ABB RobotStudio station: TransferLab2_final.rspag

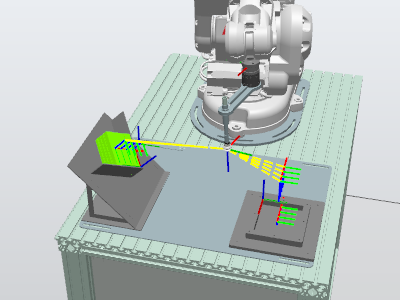
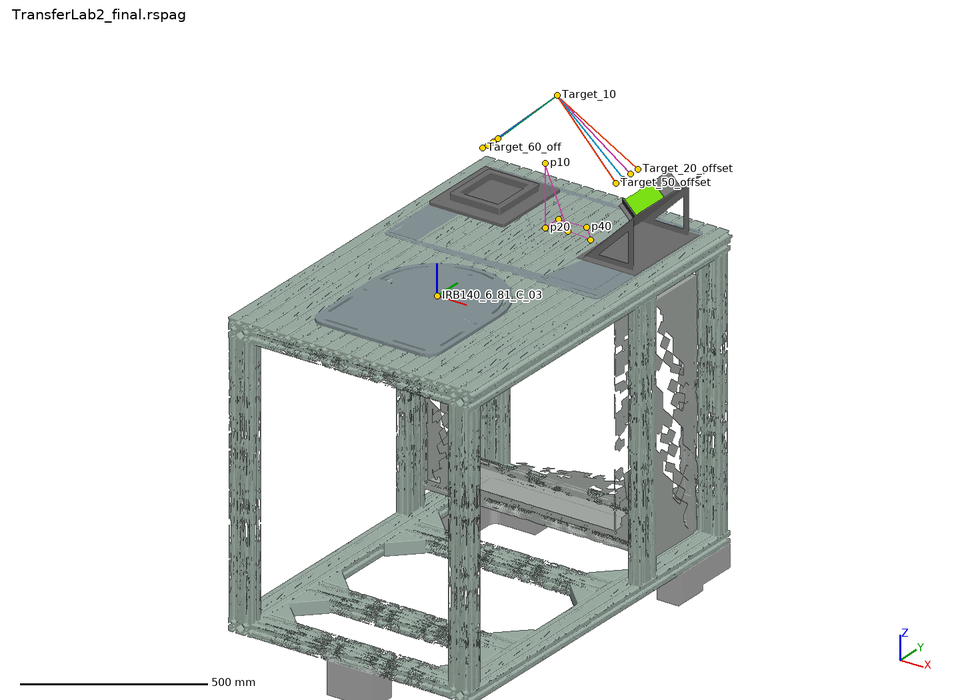
[picture v1: parts stored in the station drawn from their meshes, with robot base, taught points and paths (robot models come from the ABB library and are not in the file)]
--- station ---
Station AdvancedPickandPlace (saved by RobotStudio 24.1.10713.1)
Controller 140-107610, task T_ROB1: task frame (RAPID world) sits at (355.04, -190.94, 920) mm, rotated rx 0 ry 0 rz 90 deg in the station
Controller 140-107610
  mechanical unit ROB_1: IRB140_6_81_C_03, 6 joints, base frame (0, 0, 0) mm
Layout (positions relative to the parent item):
  - IRB140_6_81_C_03 [mechanism, from %ABB.RobotStudio.Models.IRB140%\IRB140_6_81_C_G_03.rslib] at (355.04, -190.94, 920) mm, rotated rx 0 ry 0 rz 90 deg; joint values [0.1928, 0.3139, 0.0677, 0.0702, 1.1676, -2.716] (rad or m)
  - Tpencil_2 [mechanism, from Libraries\Tpencil.rslib] at (0, 0, 0) mm
  - Modul_Base.prt [part], size 803.5 x 1200 x 1040 mm
  - FixturV [part] at (133.21, 403.34, 913) mm, size 245 x 265 x 30 mm
  - SnedLager_2 [part] at (709.45, 222.16, 913) mm, rotated rx 0 ry 0 rz 90 deg, size 300.2 x 214.3 x 218.7 mm
  - IRC5_Singel-Cabinet_2 [part, from %ABB.RobotStudio.Models.IRC5%\IRC5_Single-Cabinet.rslib] at (506.33, -200.93, 45.49) mm, rotated rx 90 ry 0 rz 90 deg
  - AE 1077.500 (2) [part] at (361.97, 363.55, 68.84) mm, rotated rx 90 ry 0 rz 180 deg, size 760 x 760 x 217 mm
  - tVacuum [mechanism, from Libraries\tVacuum.rslib] at (248.37, 333.62, 1408.02) mm, rotated rx -176.11 ry 0.46 rz 75.14 deg
  - SmartComponent_1 [smart component]
    - Source [smart component, from Components\Source.rslib]
        properties: Source=(none); Copy=cuboid_black_16; Parent=(none); Position=[0 0 0]; Orientation=[0 0 0]; Transient=false; PhysicsBehavior=0
  - cuboid_black_1 [part] at (1319.88, -207.47, 357.2) mm, rotated rx -33.6 ry -27.27 rz 53.23 deg, size 23.4 x 118 x 15.7 mm
  - cuboid_black_2 [part] at (1331.4, -191.2, 368.68) mm, rotated rx -33.6 ry -27.27 rz 53.23 deg, size 23.4 x 118 x 15.7 mm
  - cuboid_black_3 [part] at (1342.92, -174.94, 380.16) mm, rotated rx -33.6 ry -27.27 rz 53.23 deg, size 23.4 x 118 x 15.7 mm
  - cuboid_black_4 [part] at (1354.44, -158.68, 391.64) mm, rotated rx -33.6 ry -27.27 rz 53.23 deg, size 23.4 x 118 x 15.7 mm
  - cuboid_black_5 [part] at (1310.35, -207.47, 366.76) mm, rotated rx -33.6 ry -27.27 rz 53.23 deg, size 23.4 x 118 x 15.7 mm
  - cuboid_black_6 [part] at (1321.87, -191.2, 378.24) mm, rotated rx -33.6 ry -27.27 rz 53.23 deg, size 23.4 x 118 x 15.7 mm
  - cuboid_black_7 [part] at (1333.39, -174.94, 389.72) mm, rotated rx -33.6 ry -27.27 rz 53.23 deg, size 23.4 x 118 x 15.7 mm
  - cuboid_black_8 [part] at (1344.91, -158.68, 401.2) mm, rotated rx -33.6 ry -27.27 rz 53.23 deg, size 23.4 x 118 x 15.7 mm
  - cuboid_black_9 [part] at (1300.82, -207.47, 376.32) mm, rotated rx -33.6 ry -27.27 rz 53.23 deg, size 23.4 x 118 x 15.7 mm
  - cuboid_black_10 [part] at (1312.34, -191.2, 387.8) mm, rotated rx -33.6 ry -27.27 rz 53.23 deg, size 23.4 x 118 x 15.7 mm
  - cuboid_black_11 [part] at (1323.86, -174.94, 399.28) mm, rotated rx -33.6 ry -27.27 rz 53.23 deg, size 23.4 x 118 x 15.7 mm
  - cuboid_black_12 [part] at (1335.38, -158.68, 410.76) mm, rotated rx -33.6 ry -27.27 rz 53.23 deg, size 23.4 x 118 x 15.7 mm
  - cuboid_black_13 [part] at (1295.8, -202.6, 389.58) mm, rotated rx -33.76 ry -27.57 rz 53.58 deg, size 23.4 x 118 x 15.7 mm
  - cuboid_black_14 [part] at (1302.81, -191.2, 397.36) mm, rotated rx -33.6 ry -27.27 rz 53.23 deg, size 23.4 x 118 x 15.7 mm
  - cuboid_black_15 [part] at (1314.33, -174.94, 408.84) mm, rotated rx -33.6 ry -27.27 rz 53.23 deg, size 23.4 x 118 x 15.7 mm
  - cuboid_black_16 [part] at (1325.85, -158.68, 420.32) mm, rotated rx -33.6 ry -27.27 rz 53.23 deg, size 23.4 x 118 x 15.7 mm
  - RobotFrame [frame] at (355.04, -263.33, 920) mm, rotated rx 0 ry 0 rz 90 deg
Attachment: tVacuum is attached to IRB140_6_81_C_03 / Link6
Attachment: DropBox is attached to FixturV
Attachment: InclinedPickupBox is attached to SnedLager_2
Attachment: WobjTable is attached to Modul_Base.prt
EventTableEntry 1817: Group=, Trigger=doValve1 1818, Actions=[EventTableActionAttach 1819], Comment=, ActivationMode=2, Cyclic=false
EventTableTriggerIO 1818: IOValue=[1], IRC5Controller=? -1, Operator=0, SignalSource=140-107610 514
EventTableActionAttach 1819: AttachmentParent=tVacuum 1615, AttachmentChild=? -1, MountObject=false, Offset=[X=1, Y=0, Z=0, W=0, X=0, Y=1, Z=0, W=0, X=0, Y=0, Z=1, W=0, X=0, Y=0, Z=0, W=1], FlangeIndext=0, FindNearest=true
EventTableEntry 1820: Group=, Trigger=doValve1 1821, Actions=[EventTableActionDetach 1822], Comment=, ActivationMode=2, Cyclic=false
EventTableTriggerIO 1821: IOValue=[0], IRC5Controller=? -1, Operator=0, SignalSource=140-107610 514
EventTableActionDetach 1822: AttachmentParent=tVacuum 1615, AttachmentChild=? -1

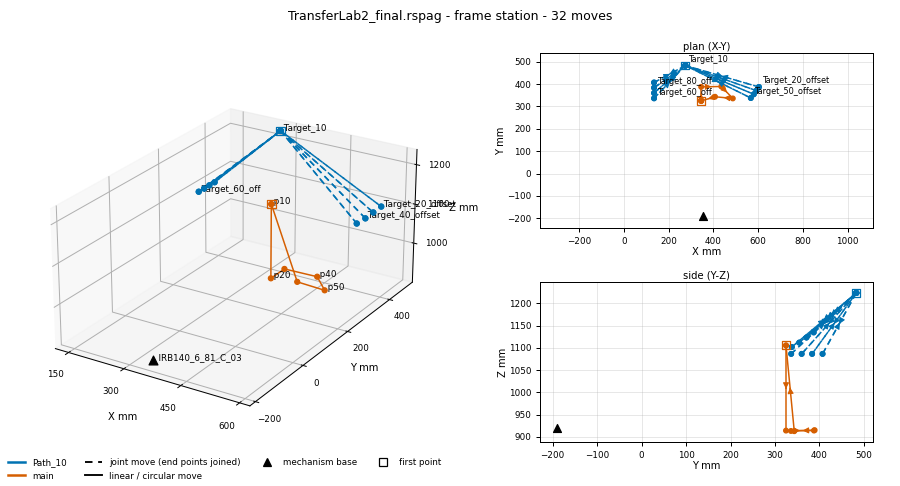
[picture p0: tool path of TransferLab2_final.rspag in frame station, 32 of 40 moves have a stored position in this frame; points joined in program order, loops and branches not executed]
--- Backups/140-107610/RAPID/TASK1/PROGMOD/MainModule.mod ---
MODULE MainModule
    PERS tooldata tVacuum:=[TRUE,[[152.46,0,183.744],[0,0,0,1]],[1.1,[1.547,-22.709,50.681],[1,0,0,0],0,0,0]];
    TASK PERS wobjdata WobjTable:=[FALSE,TRUE,"",[[280.944,-314.407,-7],[1,0,0,0]],[[0,0,0],[1,0,0,0]]];
    TASK PERS wobjdata InclinedPickupBox:=[FALSE,TRUE,"",[[562.907,-210.848,111.898],[0.35368,-0.146141,-0.352817,-0.853858]],[[0,0,0],[1,0,0,0]]];
    TASK PERS wobjdata DropBox:=[FALSE,TRUE,"",[[511.185,160.593,23],[1,0,0,0]],[[0,0,0],[1,0,0,0]]];
    !VAR intnum offset:= 14;
    !VAR intnum offset_z1;
    !VAR intnum offset_z2;
    PERS num countar :=1;



    PROC main()

        !FOR i  FROM 1 TO 5 DO
        !    offset :=14 * (i-1);
        !    offset_z1 := offset;
        !    offset_z2 := -1*offset;
        !ENDFOR

        Path_10;

    ENDPROC
ENDMODULE

--- Backups/140-107610/RAPID/TASK1/PROGMOD/Module1.mod ---
MODULE Module1
    CONST robtarget Target_10:=[[392.746094687,394.395276099,310.477856879],[0.000402904,0.129403902,0.991003532,0.034153585],[0,0,-2,0],[9E+09,9E+09,9E+09,9E+09,9E+09,9E+09]];

    CONST robtarget Target_20:=[[59.031543878,80.602128805,-4.00271589],[0.008197421,0.716388228,-0.697647201,-0.003015209],[-1,-1,-1,0],[9E+09,9E+09,9E+09,9E+09,9E+09,9E+09]];
    CONST robtarget Target_30:=[[59.031199796,57.602433832,-4.002496965],[0.008197421,0.716388228,-0.697647201,-0.003015209],[0,-1,-1,0],[9E+09,9E+09,9E+09,9E+09,9E+09,9E+09]];
    CONST robtarget Target_40:=[[59.031063684,34.601532617,-4.002986367],[0.008197421,0.716388228,-0.697647201,-0.003015209],[0,-1,-1,0],[9E+09,9E+09,9E+09,9E+09,9E+09,9E+09]];
    CONST robtarget Target_50:=[[59.260679093,11.297227236,-1.68849431],[0.008197421,0.716388228,-0.697647201,-0.003015209],[0,-1,-1,0],[9E+09,9E+09,9E+09,9E+09,9E+09,9E+09]];
    CONST robtarget Target_20_offset:=[[59.819440683,80.979027184,45.98965519],[0.008197421,0.716388228,-0.697647201,-0.003015209],[-1,-1,-1,0],[9E+09,9E+09,9E+09,9E+09,9E+09,9E+09]];
    CONST robtarget Target_30_offset:=[[59.819096601,57.979332211,45.989874115],[0.008197421,0.716388228,-0.697647201,-0.003015209],[0,-1,-1,0],[9E+09,9E+09,9E+09,9E+09,9E+09,9E+09]];
    CONST robtarget Target_40_offset:=[[59.818960489,34.978430996,45.989384713],[0.008197421,0.716388228,-0.697647201,-0.003015209],[-1,-1,-1,0],[9E+09,9E+09,9E+09,9E+09,9E+09,9E+09]];
    CONST robtarget Target_50_offset:=[[60.048575898,11.674125615,48.30387677],[0.008197421,0.716388228,-0.697647201,-0.003015209],[0,-1,-1,0],[9E+09,9E+09,9E+09,9E+09,9E+09,9E+09]];

    CONST robtarget Target_60:=[[16.076668507,59.018,-6.54],[0,0,1,0],[0,0,-2,0],[9E+09,9E+09,9E+09,9E+09,9E+09,9E+09]];
    CONST robtarget Target_60_off:=[[16.076668507,59.018,143.46],[0,0,1,0],[0,0,-2,0],[9E+09,9E+09,9E+09,9E+09,9E+09,9E+09]];
    CONST robtarget Target_70:=[[39.676668507,59.018,-6.54],[0,0,1,0],[0,0,-2,0],[9E+09,9E+09,9E+09,9E+09,9E+09,9E+09]];
    CONST robtarget Target_70_off:=[[39.676668507,59.018,143.46],[0,0,1,0],[0,0,-2,0],[9E+09,9E+09,9E+09,9E+09,9E+09,9E+09]];
    CONST robtarget Target_80:=[[63.176668507,59.018,-6.54],[0,0,1,0],[0,0,-2,0],[9E+09,9E+09,9E+09,9E+09,9E+09,9E+09]];
    CONST robtarget Target_80_off:=[[63.176668507,59.018,143.46],[0,0,1,0],[0,0,-2,0],[9E+09,9E+09,9E+09,9E+09,9E+09,9E+09]];
    CONST robtarget Target_90:=[[86.676668507,59.018,-6.54],[0,0,1,0],[0,0,-2,0],[9E+09,9E+09,9E+09,9E+09,9E+09,9E+09]];
    CONST robtarget Target_90_off:=[[86.676668507,59.018,143.46],[0,0,1,0],[0,0,-2,0],[9E+09,9E+09,9E+09,9E+09,9E+09,9E+09]];
    VAR intnum offset;
    VAR intnum offset_z1;
    VAR intnum offset_z2;


    PROC Path_10()

        FOR i  FROM 0 TO 3 DO
            offset :=14 * i;
            offset_z1 := -1*offset;
            offset_z2 := offset;

            MoveJ Target_10,v200,fine,tVacuum\WObj:=WobjTable;
            MoveJ Target_20_offset,v200,fine,tVacuum\WObj:=InclinedPickupBox;
            MoveJ Offs(Target_20,0,0,offset_z1),v200,fine,tVacuum\WObj:=InclinedPickupBox;
            !MoveJ Target_20,v200,fine,tVacuum\WObj:=InclinedPickupBox;
            WaitTime 0.3;
            SetDO doValve1, 1;
            WaitTime 0.3;
            MoveJ Target_20_offset,v200,fine,tVacuum\WObj:=InclinedPickupBox;
            MoveJ Target_10,v200,fine,tVacuum\WObj:=WobjTable;
            MoveJ Target_60_off,v200,fine,tVacuum\WObj:=DropBox;
            MoveJ Offs(Target_60,0,0,offset_z2),v200,fine,tVacuum\WObj:=DropBox;
            !MoveJ Target_60,v200,fine,tVacuum\WObj:=DropBox;
            WaitTime 0.3;
            SetDO doValve1, 0;
            WaitTime 0.3;
            MoveJ Target_60_off,v200,fine,tVacuum\WObj:=DropBox;

            MoveJ Target_10,v200,fine,tVacuum\WObj:=WobjTable;
            MoveJ Target_30_offset,v200,fine,tVacuum\WObj:=InclinedPickupBox;
            MoveJ Offs(Target_30,0,0,offset_z1),v200,fine,tVacuum\WObj:=InclinedPickupBox;
            WaitTime 0.3;
            SetDO doValve1, 1;
            WaitTime 0.3;
            MoveJ Target_30_offset,v200,fine,tVacuum\WObj:=InclinedPickupBox;
            MoveJ Target_10,v200,fine,tVacuum\WObj:=WobjTable;
            MoveJ Target_70_off,v200,fine,tVacuum\WObj:=DropBox;
            MoveJ Offs(Target_70,0,0,offset_z2),v200,fine,tVacuum\WObj:=DropBox;
            WaitTime 0.3;
            SetDO doValve1, 0;
            WaitTime 0.3;
            MoveJ Target_70_off,v200,fine,tVacuum\WObj:=DropBox;

            MoveJ Target_10,v200,fine,tVacuum\WObj:=WobjTable;
            MoveJ Target_40_offset,v200,fine,tVacuum\WObj:=InclinedPickupBox;
            MoveJ Offs(Target_40,0,0,offset_z1),v200,fine,tVacuum\WObj:=InclinedPickupBox;
            WaitTime 0.3;
            SetDO doValve1, 1;
            WaitTime 0.3;
            MoveJ Target_40_offset,v200,fine,tVacuum\WObj:=InclinedPickupBox;
            MoveJ Target_10,v200,fine,tVacuum\WObj:=WobjTable;
            MoveJ Target_80_off,v200,fine,tVacuum\WObj:=DropBox;
            MoveJ Offs(Target_80,0,0,offset_z2),v200,fine,tVacuum\WObj:=DropBox;
            WaitTime 0.3;
            SetDO doValve1, 0;
            WaitTime 0.3;
            MoveJ Target_80_off,v200,fine,tVacuum\WObj:=DropBox;

            MoveJ Target_10,v200,fine,tVacuum\WObj:=WobjTable;
            MoveJ Target_50_offset,v200,fine,tVacuum\WObj:=InclinedPickupBox;
            MoveJ Offs(Target_50,0,0,offset_z1),v200,fine,tVacuum\WObj:=InclinedPickupBox;
            WaitTime 0.3;
            SetDO doValve1, 1;
            WaitTime 0.3;
            MoveJ Target_50_offset,v200,fine,tVacuum\WObj:=InclinedPickupBox;
            MoveJ Target_10,v200,fine,tVacuum\WObj:=WobjTable;
            MoveJ Target_90_off,v200,fine,tVacuum\WObj:=DropBox;
            MoveJ Offs(Target_90,0,0,offset_z2),v200,fine,tVacuum\WObj:=DropBox;
            WaitTime 0.3;
            SetDO doValve1, 0;
            WaitTime 0.3;
            MoveJ Target_90_off,v200,fine,tVacuum\WObj:=DropBox;
            MoveJ Target_10,v200,fine,tVacuum\WObj:=WobjTable;

        ENDFOR


    ENDPROC
ENDMODULE

--- Backups/140-107610/HOME/wobj1/MainModule.mod ---
MODULE MainModule
	PERS tooldata tpencil:=[TRUE,[[-158.365,-2.10512,218.153],[1,0,0,0]],[0.5,[0,50,20],[1,0,0,0],0,0,0]];
	CONST robtarget p10:=[[515.61,9.13,185.47],[0.0619205,-0.079314,-0.994803,-0.0155883],[0,0,4,0],[9E+09,9E+09,9E+09,9E+09,9E+09,9E+09]];
	CONST robtarget p20:=[[515.61,9.13,-6.06],[0.0619228,-0.0793163,-0.994802,-0.0155846],[0,0,4,0],[9E+09,9E+09,9E+09,9E+09,9E+09,9E+09]];
	CONST robtarget p30:=[[578.43,9.13,-5.93],[0.0619495,-0.0792905,-0.994803,-0.015573],[0,0,4,0],[9E+09,9E+09,9E+09,9E+09,9E+09,9E+09]];
	CONST robtarget p40:=[[580.05,-80.82,-5.11],[0.0619285,-0.0793003,-0.994803,-0.0155876],[-1,0,3,0],[9E+09,9E+09,9E+09,9E+09,9E+09,9E+09]];
	CONST robtarget p50:=[[526.72,-132.09,-6.90],[0.0619458,-0.0792925,-0.994803,-0.0155861],[-1,0,3,0],[9E+09,9E+09,9E+09,9E+09,9E+09,9E+09]];
	CONST robtarget p60:=[[534.19,-52.76,-7.42],[0.0619566,-0.0792931,-0.994802,-0.015582],[-1,0,4,0],[9E+09,9E+09,9E+09,9E+09,9E+09,9E+09]];
	CONST robtarget p80:=[[533.93,-53.00,-9.15],[0.0619823,-0.0792257,-0.994806,-0.0155703],[-1,0,4,0],[9E+09,9E+09,9E+09,9E+09,9E+09,9E+09]];
	TASK PERS wobjdata wobj1:=[FALSE,TRUE,"",[[437.294,-191.242,-5.21685],[0.999806,-0.00979503,0.0148767,0.00835695]],[[0,0,0],[1,0,0,0]]];
	TASK PERS wobjdata wobj2:=[FALSE,TRUE,"",[[560.405,50.3251,-9.50006],[0.999834,0.00238531,-0.015124,0.00988946]],[[0,0,0],[1,0,0,0]]];
	PROC main()
		MoveJ p10, v300, fine, tpencil;
		MoveL p20, v300, fine, tpencil;
		MoveL p30, v300, fine, tpencil;
		MoveL p40, v300, fine, tpencil;
		MoveL p50, v300, fine, tpencil;
		MoveL p60, v300, fine, tpencil;
		MoveL p10, v300, fine, tpencil;
	ENDPROC
ENDMODULE

--- Backups/140-107610/SYSPAR/EIO.cfg ---
EIO:CFG_1.0:6:1::
#
SYSSIG_OUT:

      -Status "MotorOn" -Signal "doMotorLamp"

      -Status "EmStop" -Signal "doEmstopLamp"
#
INDUSTRIAL_NETWORK:

      -Name "DeviceNet" -Label "DeviceNet Master/Slave Network" -Address "2"

      -Name "PROFIBUS_Anybus" -Label "PROFIBUS Anybus Network" -Address "125"
#
EIO_CROSS:

      -Name "SYJ5325Control1" -Res "doSYJ5323_A" -Act1 "doValve1" -Oper1 "AND"\
      -Act2 "doYJ5123" -Act2_invert

      -Name "SYJ5323Control2" -Res "doSYJ5323_B" -Act1 "doValve1" -Act1_invert \
      -Oper1 "AND" -Act2 "doYJ5123" -Act2_invert

      -Name "SYJ5123Control" -Res "doYJ5123" -Act1 "diToolChangeButton"\
      -Oper1 "OR" -Act2 "doToolChanger"
#
ETHERNETIP_DEVICE:

      -Name "Local_IO" -VendorName "ABB Robotics" -ProductName "DSQC1030"\
      -Label "ABB Local I/O Device" -Address "192.168.125.100" -VendorId 75\
      -ProductCode 29 -DeviceType 12 -OutputAssembly 100 -InputAssembly 101\
      -ConfigurationAssembly 102 -InputConnectionType "POINT2POINT"\
      -ConnectionPriority "SCHEDULE" -OutputSize 2 -InputSize 2\
      -ConfigurationSize 8\
      -ConfigurationData00 "01 02 09 10 01 08 10 01 00 00 00 00 00 00 00 00"\
      -O2T_RPI 40000 -T2O_RPI 40000
#
DEVICENET_INTERNAL_DEVICE:

      -Name "DN_Internal_Device" -VendorName "ABB Robotics"\
      -ProductName "DeviceNet Internal Slave Device"
#
PROFIBUS_INTERNAL_ANYBUS_DEVICE:

      -Name "PB_Internal_Anybus" -VendorName "ABB Robotics"\
      -ProductName "PROFIBUS Internal Anybus Device"
#
EIO_SIGNAL:

      -Name "doToolChanger" -SignalType "DO" -DeviceMap "0"

      -Name "doSYJ5323_A" -SignalType "DO" -Device "Local_IO" -DeviceMap "1"

      -Name "doSYJ5323_B" -SignalType "DO" -Device "Local_IO" -DeviceMap "2"

      -Name "doMotorLamp" -SignalType "DO" -Device "Local_IO" -DeviceMap "3"

      -Name "do1RobotContact" -SignalType "DO" -Device "Local_IO" -DeviceMap "4"

      -Name "do2RobotContact" -SignalType "DO" -Device "Local_IO" -DeviceMap "5"

      -Name "doYellowLamp" -SignalType "DO" -Device "Local_IO" -DeviceMap "6"

      -Name "doEmstopLamp" -SignalType "DO" -Device "Local_IO" -DeviceMap "7"

      -Name "Local_IO_0_DO9" -SignalType "DO" -Device "Local_IO" -DeviceMap "8"

      -Name "Local_IO_0_DO10" -SignalType "DO" -Device "Local_IO" -DeviceMap "9"

      -Name "Local_IO_0_DO11" -SignalType "DO" -Device "Local_IO"\
      -DeviceMap "10"

      -Name "Local_IO_0_DO12" -SignalType "DO" -Device "Local_IO"\
      -DeviceMap "11"

      -Name "Local_IO_0_DO13" -SignalType "DO" -Device "Local_IO"\
      -DeviceMap "12"

      -Name "Local_IO_0_DO14" -SignalType "DO" -Device "Local_IO"\
      -DeviceMap "13"

      -Name "Local_IO_0_DO15" -SignalType "DO" -Device "Local_IO"\
      -DeviceMap "14"

      -Name "Local_IO_0_DO16" -SignalType "DO" -Device "Local_IO"\
      -DeviceMap "15"

      -Name "di1RobotContact" -SignalType "DI" -Device "Local_IO" -DeviceMap "0"

      -Name "di2RobotContact" -SignalType "DI" -Device "Local_IO" -DeviceMap "1"

      -Name "diOkButton" -SignalType "DI" -Device "Local_IO" -DeviceMap "2"

      -Name "diToolChangeButton" -SignalType "DI" -Device "Local_IO"\
      -DeviceMap "3"

      -Name "Local_IO_0_DI5" -SignalType "DI" -Device "Local_IO" -DeviceMap "4"

      -Name "Local_IO_0_DI6" -SignalType "DI" -Device "Local_IO" -DeviceMap "5"

      -Name "Local_IO_0_DI7" -SignalType "DI" -Device "Local_IO" -DeviceMap "6"

      -Name "Local_IO_0_DI8" -SignalType "DI" -Device "Local_IO" -DeviceMap "7"

      -Name "Local_IO_0_DI9" -SignalType "DI" -Device "Local_IO" -DeviceMap "8"

      -Name "Local_IO_0_DI10" -SignalType "DI" -Device "Local_IO" -DeviceMap "9"

      -Name "Local_IO_0_DI11" -SignalType "DI" -Device "Local_IO"\
      -DeviceMap "10"

      -Name "Local_IO_0_DI12" -SignalType "DI" -Device "Local_IO"\
      -DeviceMap "11"

      -Name "Local_IO_0_DI13" -SignalType "DI" -Device "Local_IO"\
      -DeviceMap "12"

      -Name "Local_IO_0_DI14" -SignalType "DI" -Device "Local_IO"\
      -DeviceMap "13"

      -Name "Local_IO_0_DI15" -SignalType "DI" -Device "Local_IO"\
      -DeviceMap "14"

      -Name "Local_IO_0_DI16" -SignalType "DI" -Device "Local_IO"\
      -DeviceMap "15"

      -Name "doValve1" -SignalType "DO"\
      -Label "Controll of Valve1 (tool funtion)"

      -Name "doYJ5123" -SignalType "DO" -Device "Local_IO" -DeviceMap "0"
